ABB RobotStudio station: save_station_20180824-091246.rsstn

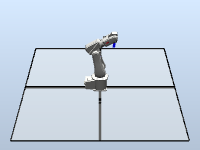
Station Station (saved by RobotStudio 6.7.7936.1011)
Controller WILL4230
  mechanical unit ROB_1: IRB120_3_58__01, 6 joints, base frame (0, 0, 0) mm
Layout (positions relative to the parent item):
  - IRB120_3_58__01 [mechanism, from Robots\IRB120_3_58_G_01.rslib] at (0, 0, 0) mm; joint values [0, -0.1947, -0.3256, 0, 2.0911, 0] (rad or m)
